REGION Network 132: EM2 cmStatus
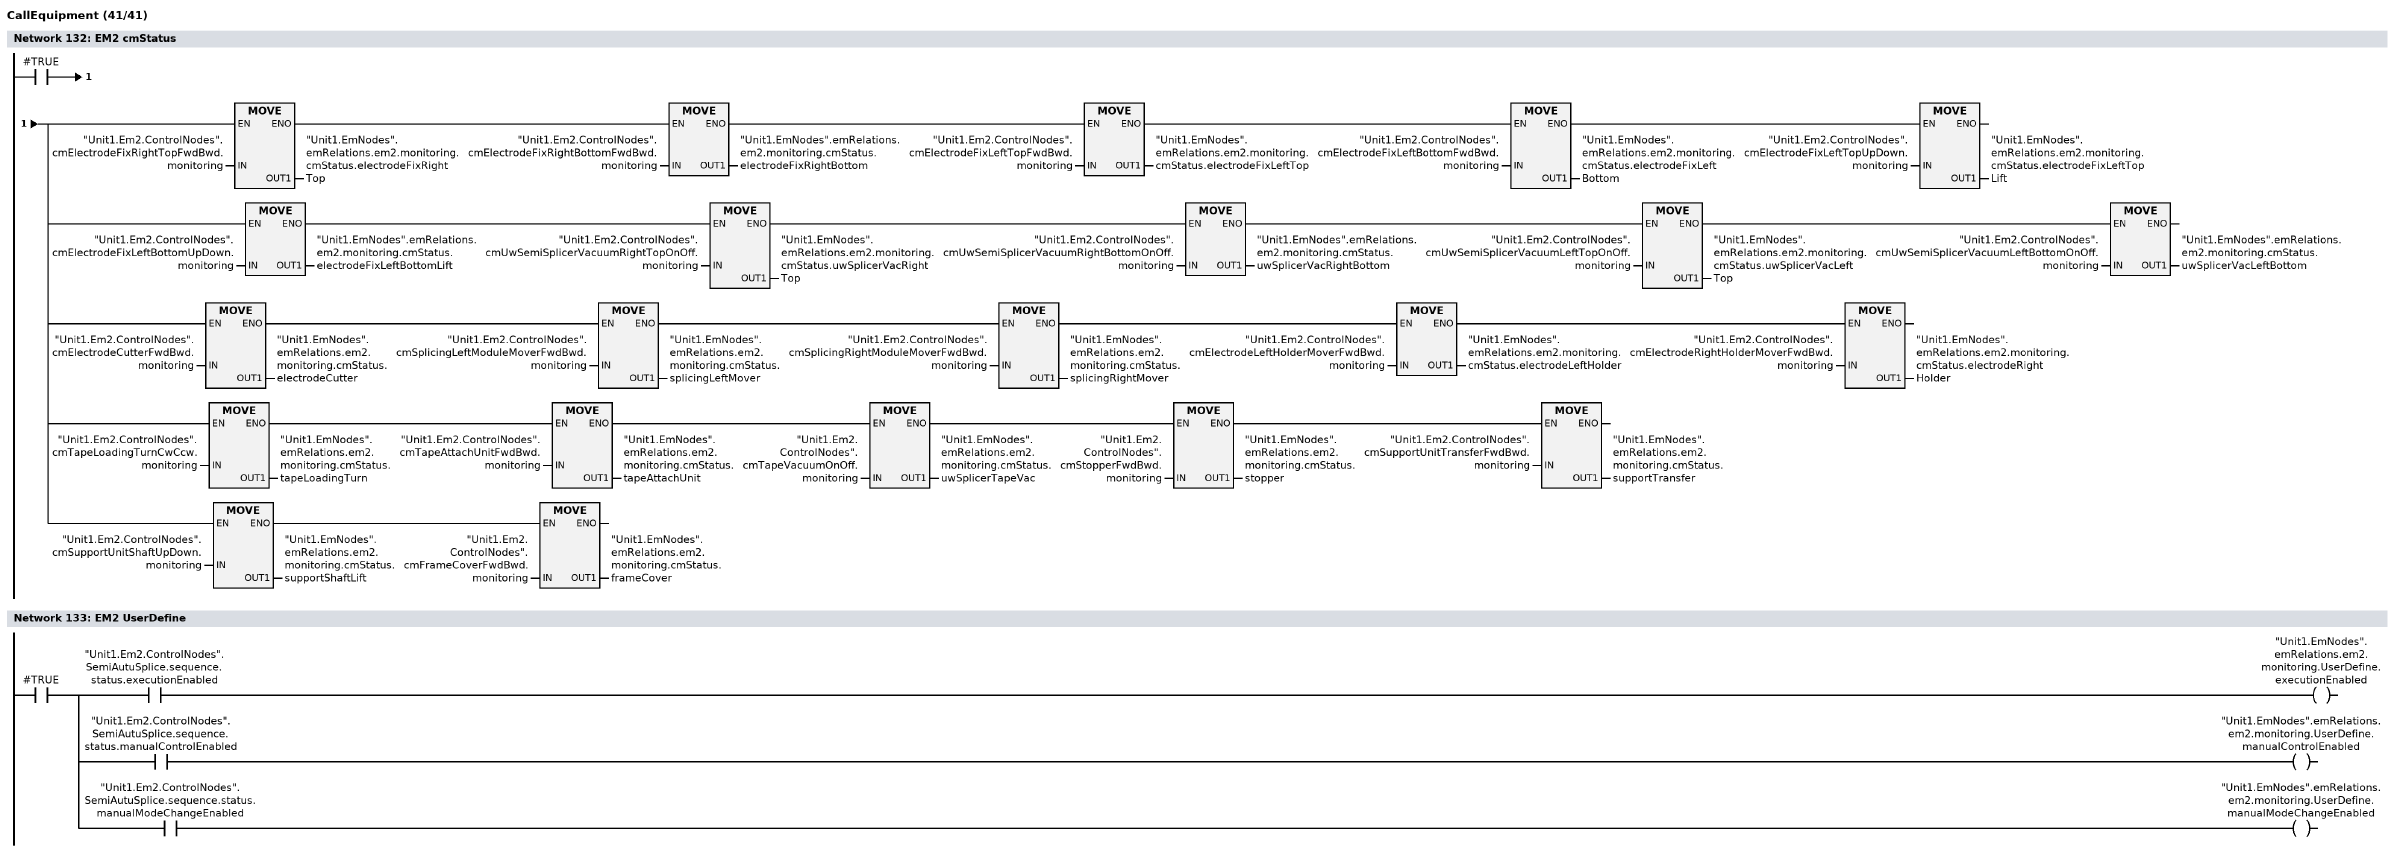
   RUNG wire#powerrail
      Contact( #TRUE )
      wire#w1
      Move(in := "Unit1.Em2.ControlNodes".cmElectrodeFixRightTopFwdBwd.monitoring, out1 => "Unit1.EmNodes".emRelations.em2.monitoring.cmStatus.electrodeFixRightTop)
      Move(in := "Unit1.Em2.ControlNodes".cmElectrodeFixRightBottomFwdBwd.monitoring, out1 => "Unit1.EmNodes".emRelations.em2.monitoring.cmStatus.electrodeFixRightBottom)
      Move(in := "Unit1.Em2.ControlNodes".cmElectrodeFixLeftTopFwdBwd.monitoring, out1 => "Unit1.EmNodes".emRelations.em2.monitoring.cmStatus.electrodeFixLeftTop)
      Move(in := "Unit1.Em2.ControlNodes".cmElectrodeFixLeftBottomFwdBwd.monitoring, out1 => "Unit1.EmNodes".emRelations.em2.monitoring.cmStatus.electrodeFixLeftBottom)
      Move(in := "Unit1.Em2.ControlNodes".cmElectrodeFixLeftTopUpDown.monitoring, out1 => "Unit1.EmNodes".emRelations.em2.monitoring.cmStatus.electrodeFixLeftTopLift)
   END_RUNG
   RUNG wire#w1
      Move(in := "Unit1.Em2.ControlNodes".cmElectrodeFixLeftBottomUpDown.monitoring, out1 => "Unit1.EmNodes".emRelations.em2.monitoring.cmStatus.electrodeFixLeftBottomLift)
      Move(in := "Unit1.Em2.ControlNodes".cmUwSemiSplicerVacuumRightTopOnOff.monitoring, out1 => "Unit1.EmNodes".emRelations.em2.monitoring.cmStatus.uwSplicerVacRightTop)
      Move(in := "Unit1.Em2.ControlNodes".cmUwSemiSplicerVacuumRightBottomOnOff.monitoring, out1 => "Unit1.EmNodes".emRelations.em2.monitoring.cmStatus.uwSplicerVacRightBottom)
      Move(in := "Unit1.Em2.ControlNodes".cmUwSemiSplicerVacuumLeftTopOnOff.monitoring, out1 => "Unit1.EmNodes".emRelations.em2.monitoring.cmStatus.uwSplicerVacLeftTop)
      Move(in := "Unit1.Em2.ControlNodes".cmUwSemiSplicerVacuumLeftBottomOnOff.monitoring, out1 => "Unit1.EmNodes".emRelations.em2.monitoring.cmStatus.uwSplicerVacLeftBottom)
   END_RUNG
   RUNG wire#w1
      Move(in := "Unit1.Em2.ControlNodes".cmElectrodeCutterFwdBwd.monitoring, out1 => "Unit1.EmNodes".emRelations.em2.monitoring.cmStatus.electrodeCutter)
      Move(in := "Unit1.Em2.ControlNodes".cmSplicingLeftModuleMoverFwdBwd.monitoring, out1 => "Unit1.EmNodes".emRelations.em2.monitoring.cmStatus.splicingLeftMover)
      Move(in := "Unit1.Em2.ControlNodes".cmSplicingRightModuleMoverFwdBwd.monitoring, out1 => "Unit1.EmNodes".emRelations.em2.monitoring.cmStatus.splicingRightMover)
      Move(in := "Unit1.Em2.ControlNodes".cmElectrodeLeftHolderMoverFwdBwd.monitoring, out1 => "Unit1.EmNodes".emRelations.em2.monitoring.cmStatus.electrodeLeftHolder)
      Move(in := "Unit1.Em2.ControlNodes".cmElectrodeRightHolderMoverFwdBwd.monitoring, out1 => "Unit1.EmNodes".emRelations.em2.monitoring.cmStatus.electrodeRightHolder)
   END_RUNG
   RUNG wire#w1
      Move(in := "Unit1.Em2.ControlNodes".cmTapeLoadingTurnCwCcw.monitoring, out1 => "Unit1.EmNodes".emRelations.em2.monitoring.cmStatus.tapeLoadingTurn)
      Move(in := "Unit1.Em2.ControlNodes".cmTapeAttachUnitFwdBwd.monitoring, out1 => "Unit1.EmNodes".emRelations.em2.monitoring.cmStatus.tapeAttachUnit)
      Move(in := "Unit1.Em2.ControlNodes".cmTapeVacuumOnOff.monitoring, out1 => "Unit1.EmNodes".emRelations.em2.monitoring.cmStatus.uwSplicerTapeVac)
      Move(in := "Unit1.Em2.ControlNodes".cmStopperFwdBwd.monitoring, out1 => "Unit1.EmNodes".emRelations.em2.monitoring.cmStatus.stopper)
      Move(in := "Unit1.Em2.ControlNodes".cmSupportUnitTransferFwdBwd.monitoring, out1 => "Unit1.EmNodes".emRelations.em2.monitoring.cmStatus.supportTransfer)
   END_RUNG
   RUNG wire#w1
      Move(in := "Unit1.Em2.ControlNodes".cmSupportUnitShaftUpDown.monitoring, out1 => "Unit1.EmNodes".emRelations.em2.monitoring.cmStatus.supportShaftLift)
      Move(in := "Unit1.Em2.ControlNodes".cmFrameCoverFwdBwd.monitoring, out1 => "Unit1.EmNodes".emRelations.em2.monitoring.cmStatus.frameCover)
   END_RUNG
   // the same network as SCL:
   IF #TRUE THEN
       "Unit1.EmNodes".emRelations.em2.monitoring.cmStatus.electrodeFixRightTop := "Unit1.Em2.ControlNodes".cmElectrodeFixRightTopFwdBwd.monitoring;
       "Unit1.EmNodes".emRelations.em2.monitoring.cmStatus.electrodeFixRightBottom := "Unit1.Em2.ControlNodes".cmElectrodeFixRightBottomFwdBwd.monitoring;
       "Unit1.EmNodes".emRelations.em2.monitoring.cmStatus.electrodeFixLeftTop := "Unit1.Em2.ControlNodes".cmElectrodeFixLeftTopFwdBwd.monitoring;
       "Unit1.EmNodes".emRelations.em2.monitoring.cmStatus.electrodeFixLeftBottom := "Unit1.Em2.ControlNodes".cmElectrodeFixLeftBottomFwdBwd.monitoring;
       "Unit1.EmNodes".emRelations.em2.monitoring.cmStatus.electrodeFixLeftTopLift := "Unit1.Em2.ControlNodes".cmElectrodeFixLeftTopUpDown.monitoring;
       "Unit1.EmNodes".emRelations.em2.monitoring.cmStatus.electrodeFixLeftBottomLift := "Unit1.Em2.ControlNodes".cmElectrodeFixLeftBottomUpDown.monitoring;
       "Unit1.EmNodes".emRelations.em2.monitoring.cmStatus.uwSplicerVacRightTop := "Unit1.Em2.ControlNodes".cmUwSemiSplicerVacuumRightTopOnOff.monitoring;
       "Unit1.EmNodes".emRelations.em2.monitoring.cmStatus.uwSplicerVacRightBottom := "Unit1.Em2.ControlNodes".cmUwSemiSplicerVacuumRightBottomOnOff.monitoring;
       "Unit1.EmNodes".emRelations.em2.monitoring.cmStatus.uwSplicerVacLeftTop := "Unit1.Em2.ControlNodes".cmUwSemiSplicerVacuumLeftTopOnOff.monitoring;
       "Unit1.EmNodes".emRelations.em2.monitoring.cmStatus.uwSplicerVacLeftBottom := "Unit1.Em2.ControlNodes".cmUwSemiSplicerVacuumLeftBottomOnOff.monitoring;
       "Unit1.EmNodes".emRelations.em2.monitoring.cmStatus.electrodeCutter := "Unit1.Em2.ControlNodes".cmElectrodeCutterFwdBwd.monitoring;
       "Unit1.EmNodes".emRelations.em2.monitoring.cmStatus.splicingLeftMover := "Unit1.Em2.ControlNodes".cmSplicingLeftModuleMoverFwdBwd.monitoring;
       "Unit1.EmNodes".emRelations.em2.monitoring.cmStatus.splicingRightMover := "Unit1.Em2.ControlNodes".cmSplicingRightModuleMoverFwdBwd.monitoring;
       "Unit1.EmNodes".emRelations.em2.monitoring.cmStatus.electrodeLeftHolder := "Unit1.Em2.ControlNodes".cmElectrodeLeftHolderMoverFwdBwd.monitoring;
       "Unit1.EmNodes".emRelations.em2.monitoring.cmStatus.electrodeRightHolder := "Unit1.Em2.ControlNodes".cmElectrodeRightHolderMoverFwdBwd.monitoring;
       "Unit1.EmNodes".emRelations.em2.monitoring.cmStatus.tapeLoadingTurn := "Unit1.Em2.ControlNodes".cmTapeLoadingTurnCwCcw.monitoring;
       "Unit1.EmNodes".emRelations.em2.monitoring.cmStatus.tapeAttachUnit := "Unit1.Em2.ControlNodes".cmTapeAttachUnitFwdBwd.monitoring;
       "Unit1.EmNodes".emRelations.em2.monitoring.cmStatus.uwSplicerTapeVac := "Unit1.Em2.ControlNodes".cmTapeVacuumOnOff.monitoring;
       "Unit1.EmNodes".emRelations.em2.monitoring.cmStatus.stopper := "Unit1.Em2.ControlNodes".cmStopperFwdBwd.monitoring;
       "Unit1.EmNodes".emRelations.em2.monitoring.cmStatus.supportTransfer := "Unit1.Em2.ControlNodes".cmSupportUnitTransferFwdBwd.monitoring;
       "Unit1.EmNodes".emRelations.em2.monitoring.cmStatus.supportShaftLift := "Unit1.Em2.ControlNodes".cmSupportUnitShaftUpDown.monitoring;
       "Unit1.EmNodes".emRelations.em2.monitoring.cmStatus.frameCover := "Unit1.Em2.ControlNodes".cmFrameCoverFwdBwd.monitoring;
   END_IF;
END_REGION

REGION Network 133: EM2 UserDefine
   RUNG wire#powerrail
      Contact( #TRUE )
      wire#w1
      Contact( "Unit1.Em2.ControlNodes".SemiAutuSplice.sequence.status.executionEnabled )
      Coil( "Unit1.EmNodes".emRelations.em2.monitoring.UserDefine.executionEnabled )
   END_RUNG
   RUNG wire#w1
      Contact( "Unit1.Em2.ControlNodes".SemiAutuSplice.sequence.status.manualControlEnabled )
      Coil( "Unit1.EmNodes".emRelations.em2.monitoring.UserDefine.manualControlEnabled )
   END_RUNG
   RUNG wire#w1
      Contact( "Unit1.Em2.ControlNodes".SemiAutuSplice.sequence.status.manualModeChangeEnabled )
      Coil( "Unit1.EmNodes".emRelations.em2.monitoring.UserDefine.manualModeChangeEnabled )
   END_RUNG
   // the same network as SCL:
   "Unit1.EmNodes".emRelations.em2.monitoring.UserDefine.executionEnabled := #TRUE AND "Unit1.Em2.ControlNodes".SemiAutuSplice.sequence.status.executionEnabled;
   "Unit1.EmNodes".emRelations.em2.monitoring.UserDefine.manualControlEnabled := #TRUE AND "Unit1.Em2.ControlNodes".SemiAutuSplice.sequence.status.manualControlEnabled;
   "Unit1.EmNodes".emRelations.em2.monitoring.UserDefine.manualModeChangeEnabled := #TRUE AND "Unit1.Em2.ControlNodes".SemiAutuSplice.sequence.status.manualModeChangeEnabled;
END_REGION
END_FUNCTION_BLOCK
